FUNCTION_BLOCK FB_DataBuffer
VAR_OUTPUT
	nElements: UDINT;
END_VAR
VAR
	_nDataSize: UDINT;
	
	_pWriteBuffer: POINTER TO BYTE;
	_pWriteBufferTime: POINTER TO ARRAY [1..cEntryCount] OF ULINT;
	_pReadBuffer: POINTER TO BYTE;
	_pReadBufferTime: POINTER TO ARRAY [1..cEntryCount] OF ULINT;
	
	_pBuffer1: POINTER TO BYTE;
	_aBufferTime1: ARRAY [1..cEntryCount] OF ULINT;
	_pBuffer2: POINTER TO BYTE;
	_aBufferTime2: ARRAY [1..cEntryCount] OF ULINT;
	
	_nBufferIdx: INT := 1;
	
	_nBufferEntry_Add: UDINT;
	
	_bLock: BOOL;
	
END_VAR
VAR CONSTANT
	cEntryCount: UDINT := 25;
END_VAR

METHOD FB_init : BOOL
VAR_INPUT
	bInitRetains: BOOL; // if TRUE, the retain variables are initialized (warm start / cold start)
	bInCopyCode: BOOL; // if TRUE, the instance afterwards gets moved into the copy code (online change)
	nDataSize: UDINT;
END_VAR
VAR
END_VAR
IF NOT bInCopyCode THEN
	_nDataSize:= nDataSize;
	_Init();
END_IF
END_METHOD

METHOD FB_exit : BOOL
VAR_INPUT
	bInCopyCode: BOOL; // if TRUE, the exit method is called for exiting an instance that is copied afterwards (online change).
END_VAR
VAR
END_VAR
IF _pBuffer1 <> 0 THEN
	__DELETE(_pBuffer1);
END_IF

IF _pBuffer2 <> 0 THEN
	__DELETE(_pBuffer2);
END_IF

_pWriteBuffer:= 0;
_pWriteBufferTime:= 0;
_pReadBuffer:= 0;
_pReadBufferTime:= 0;

_nBufferIdx:= 0;
_nBufferEntry_Add:= 0;
END_METHOD

METHOD PRIVATE _Init : BOOL
VAR
END_VAR
IF _pBuffer1 <> 0 THEN
	__DELETE(_pBuffer1);
END_IF

IF _pBuffer2 <> 0 THEN
	__DELETE(_pBuffer2);
END_IF

_pBuffer1 := __NEW(BYTE, (_nDataSize * cEntryCount));
_pBuffer2 := __NEW(BYTE, (_nDataSize * cEntryCount));

_nBufferIdx:= 0;

Call();
END_METHOD

METHOD Call : BOOL
VAR
END_VAR
nElements:= 0;

IF TestAndSet(_bLock) THEN

	_nBufferIdx:= _nBufferIdx + 1;
	IF _nBufferIdx >= 3 THEN
		_nBufferIdx:= 1;
	END_IF

	CASE _nBufferIdx OF
		1:
			_pWriteBuffer:= _pBuffer1;
			_pReadBuffer:= _pBuffer2;

			_pWriteBufferTime:= ADR(_aBufferTime1);
			_pReadBufferTime:= ADR(_aBufferTime2);
		2:
			_pWriteBuffer:= _pBuffer2;
			_pReadBuffer:= _pBuffer1;

			_pWriteBufferTime:= ADR(_aBufferTime2);
			_pReadBufferTime:= ADR(_aBufferTime1);
	END_CASE

	nElements:= _nBufferEntry_Add;

	_nBufferEntry_Add:= 0;
	_bLock:= FALSE;
END_IF
END_METHOD

METHOD AddData : BOOL
VAR_INPUT
	pDataIn: PVOID;
END_VAR
VAR
END_VAR
IF TestAndSet(_bLock) THEN

	IF _pWriteBuffer <> 0 AND pDataIn <> 0 THEN

		IF _nBufferEntry_Add >= cEntryCount THEN
			_nBufferEntry_Add:= cEntryCount - 1;
		END_IF

		MEMCPY(_pWriteBuffer + (_nBufferEntry_Add * _nDataSize), pDataIn, _nDataSize);

		_nBufferEntry_Add:= _nBufferEntry_Add + 1;

		IF _pWriteBufferTime <> 0 THEN
			_pWriteBufferTime^[_nBufferEntry_Add]:= F_GetActualDcTime64();
		END_IF

	END_IF

	_bLock:= FALSE;
END_IF
END_METHOD

METHOD GetData : BOOL
VAR_INPUT
	nElement: UDINT(1..cEntryCount);
	pDataOut: PVOID;
END_VAR
VAR
END_VAR
IF nElement <= nElements THEN
	IF pDataOut <> 0 AND _pReadBuffer <> 0 THEN
		MEMCPY(pDataOut, _pReadBuffer + ((nElement-1) * _nDataSize), _nDataSize);
	END_IF
END_IF
END_METHOD

METHOD GetTimestamp : ULINT
VAR_INPUT
	nElement: UDINT(1..cEntryCount);
END_VAR
VAR
END_VAR
IF _pReadBufferTime <> 0 THEN
	GetTimestamp:= _pReadBufferTime^[nElement];
END_IF
END_METHOD

END_FUNCTION_BLOCK

(* stored: POU FB_DataBuffer: Id 0c14ef56-9a09-423d-a3dd-a18323502d23, SpecialFunc None
   Method FB_init: Id 344a8027-b879-4722-8461-651fb7d5b6c6
   Method FB_exit: Id 3e1e124c-6c4a-40bd-a957-13bcd6bd02c9
   Method _Init: Id f856828b-1f9a-4a67-a44c-3c3e9e9a5437
   Method Call: Id d63a8be4-ac65-4acb-a04d-a8a5bd51843d
   Method AddData: Id 181dbe0a-318e-4b76-8866-5f3f90f8a271
   Method GetData: Id 61ac8db9-8e63-482d-905d-e0ca95e12d6b
   Method GetTimestamp: Id d3d7d746-2354-4a0b-9e47-6dd1a8942360 *)
